(*
SPDX-FileCopyrightText: © 2026 Oleksandr Tiutyk <trofimich@gmail.com>
SPDX-License-Identifier: MIT
License: https://opensource.org/license/mit
*)

INTERFACE IWorkflowElement EXTENDS IVariableContainer, TOF_Core.INamed

{attribute 'monitoring' := 'call'}
PROPERTY Parent : IWorkflowElement
GET
END_GET
END_PROPERTY

END_INTERFACE

(* stored: Version 1.1.0.1
   Itf IWorkflowElement: Id {9f2cf0e1-485a-4f9c-a99d-72fe864dad44}
   Property Parent: Id {cfa98d13-c681-4820-8998-f8a3411bc85d}
   Get Get: Id {7ec43eb9-38c8-4405-b62f-59911e7d0170} *)
